FUNCTION_BLOCK FB_MarqueeExPause EXTENDS FB_MarqueeEx
VAR_INPUT
	pPause		:POINTER TO BOOL;
	pStop		:POINTER TO BOOL;
END_VAR
VAR_OUTPUT
END_VAR
VAR
END_VAR

METHOD Blinking : BOOL
VAR_INPUT
	bStart			:BOOL;
END_VAR
VAR
	
END_VAR

IF bStart THEN 
	
	CASE iStep OF 
		0:
			pLamp01^ := TRUE;
			THIS^.Delay();
			IF THIS^.bDelayOK THEN 
				pLamp01^ := NOT pLamp01^;
				THIS^.Reset();
				iStep := 10;
			END_IF
		10:
			pLamp02^ := TRUE;
			THIS^.Delay();
			IF bDelayOK THEN 
				pLamp02^ := NOT pLamp02^;
				THIS^.Reset();
				iStep := 20;
			END_IF
		20:
			pLamp03^ := TRUE;
			THIS^.Delay();
			IF bDelayOK THEN 
				pLamp03^ := NOT pLamp03^;
				THIS^.Reset();
				iStep := 30;
			END_IF
		30:
			pLamp04^ := TRUE;
			THIS^.Delay();
			IF bDelayOK THEN 
				pLamp04^ := NOT pLamp04^;
				THIS^.Reset();
				IF pStop^ THEN 
					bStart := NOT bStart;					
					//pStop^ := NOT pStop^;			
					//iStep := 0;
				ELSE
					iStep := 0;
				END_IF				
			END_IF		
	END_CASE
ELSE 
	pLamp04^ := FALSE;
	pLamp03^ := FALSE;
	pLamp02^ := FALSE;
	pLamp01^ := FALSE;
END_IF
END_METHOD

METHOD Delay : BOOL
VAR_INPUT
END_VAR
CASE iDelayStep OF
	0:
		bDelayOK := FALSE;
		TON1(IN:=FALSE);		 
		iDelayStep := 10;
	10:
		TON1(IN:=TRUE , PT:= pTime^, Q=> , ET=> );
		IF TON1.Q THEN 						
			IF NOT pPause^  THEN
				TON1(IN:=FALSE);
				bDelayOK := TRUE;
				iDelayStep := 100;
			END_IF
			
		END_IF
END_CASE
END_METHOD

END_FUNCTION_BLOCK

(* stored: Version 1.1.0.1, ProductVersion 3.1.4022.16
   POU FB_MarqueeExPause: Id {e94b50f9-9adc-4792-ab78-0997689169a6}, SpecialFunc None
   Method Blinking: Id {d0efd987-3dd9-4ae1-bf7b-aefa7766ca45}
   Method Delay: Id {bbf514b6-5e0c-4e1b-b098-02a940d7e096} *)
